REGION Network 114: NG_1
   RUNG wire#powerrail
      Contact( "AlwaysTRUE" )
      wire#w1
      Contact( "PalletNGData".LoadingNGPallet.NG_2_1 )
      Contact( "PalletNGData".LoadingNGPallet.NG_2_2 )
      Contact( "PalletNGData".LoadingNGPallet.NG_2_3 )
      Contact( "PalletNGData".LoadingNGPallet.NG_2_4 )
      Contact( "PalletNGData".LoadingNGPallet.NG_2_5 )
      { S7_Templates := "time_type := Time" } "TON".TON[50].TON(pt := t#4s, et =>)
      Coil( "ST10_DeviceError"."E".NG_1.ShaftScanNGFull )
   END_RUNG
   RUNG wire#w1
      Contact( "PalletNGData".LoadingNGPallet.NG_1_1 )
      Contact( "PalletNGData".LoadingNGPallet.NG_1_2 )
      Contact( "PalletNGData".LoadingNGPallet.NG_1_3 )
      Contact( "PalletNGData".LoadingNGPallet.NG_1_4 )
      Contact( "PalletNGData".LoadingNGPallet.NG_1_5 )
      { S7_Templates := "time_type := Time" } "TON".TON[51].TON(pt := t#4s, et =>)
      Coil( "ST10_DeviceError"."E".NG_1.PressNGFull )
   END_RUNG
   RUNG wire#w1
      Contact( "PalletNGData".LoadingNGPallet.NG_3_1 )
      Contact( "PalletNGData".LoadingNGPallet.NG_3_2 )
      Contact( "PalletNGData".LoadingNGPallet.NG_3_3 )
      Contact( "PalletNGData".LoadingNGPallet.NG_3_4 )
      Contact( "PalletNGData".LoadingNGPallet.NG_3_5 )
      { S7_Templates := "time_type := Time" } "TON".TON[52].TON(pt := t#4s, et =>)
      Coil( "ST10_DeviceError"."E".NG_1.RingScanNGFull )
   END_RUNG
   RUNG wire#w1
      I_Contact( "PalletNGData".LoadingNGPallet.Ready_1 )
      Contact( "Station_Sys".Auto.Mode )
      I_Contact( "KukaRobot1_CtrlDB".sROBtoPLC.User.Cycle.DO225_ScanPosInside )
      I_Contact( "KukaRobot1_CtrlDB".sROBtoPLC.User.Cycle.DO265_LoadNGInside )
      { S7_Templates := "time_type := Time" } "TON".TON[53].TON(pt := t#4s, et =>)
      I_Contact( true )
      Coil( "ST10_DeviceError"."E".NG_1.ShaftScanStatus )
   END_RUNG
   RUNG wire#w1
      I_Contact( "PalletNGData".LoadingNGPallet.Ready_2 )
      Contact( "Station_Sys".Auto.Mode )
      I_Contact( "KukaRobot1_CtrlDB".sROBtoPLC.User.Cycle.DO225_ScanPosInside )
      I_Contact( "KukaRobot1_CtrlDB".sROBtoPLC.User.Cycle.DO265_LoadNGInside )
      { S7_Templates := "time_type := Time" } "TON".TON[54].TON(pt := t#4s, et =>)
      I_Contact( true )
      Coil( "ST10_DeviceError"."E".NG_1.PressNGStatus )
   END_RUNG
   RUNG wire#w1
      I_Contact( "PalletNGData".LoadingNGPallet.Ready_3 )
      Contact( "Station_Sys".Auto.Mode )
      I_Contact( "KukaRobot1_CtrlDB".sROBtoPLC.User.Cycle.DO225_ScanPosInside )
      I_Contact( "KukaRobot1_CtrlDB".sROBtoPLC.User.Cycle.DO265_LoadNGInside )
      { S7_Templates := "time_type := Time" } "TON".TON[55].TON(pt := t#4s, et =>)
      I_Contact( true )
      Coil( "ST10_DeviceError"."E".NG_1.RingScanNGStatus )
   END_RUNG
   // the same network as SCL:
   "TON".TON[50].TON(IN := "AlwaysTRUE" AND "PalletNGData".LoadingNGPallet.NG_2_1 AND "PalletNGData".LoadingNGPallet.NG_2_2 AND "PalletNGData".LoadingNGPallet.NG_2_3 AND "PalletNGData".LoadingNGPallet.NG_2_4 AND "PalletNGData".LoadingNGPallet.NG_2_5,
                     PT := t#4s);
   "ST10_DeviceError"."E".NG_1.ShaftScanNGFull := "TON".TON[50].Q;
   "TON".TON[51].TON(IN := "AlwaysTRUE" AND "PalletNGData".LoadingNGPallet.NG_1_1 AND "PalletNGData".LoadingNGPallet.NG_1_2 AND "PalletNGData".LoadingNGPallet.NG_1_3 AND "PalletNGData".LoadingNGPallet.NG_1_4 AND "PalletNGData".LoadingNGPallet.NG_1_5,
                     PT := t#4s);
   "ST10_DeviceError"."E".NG_1.PressNGFull := "TON".TON[51].Q;
   "TON".TON[52].TON(IN := "AlwaysTRUE" AND "PalletNGData".LoadingNGPallet.NG_3_1 AND "PalletNGData".LoadingNGPallet.NG_3_2 AND "PalletNGData".LoadingNGPallet.NG_3_3 AND "PalletNGData".LoadingNGPallet.NG_3_4 AND "PalletNGData".LoadingNGPallet.NG_3_5,
                     PT := t#4s);
   "ST10_DeviceError"."E".NG_1.RingScanNGFull := "TON".TON[52].Q;
   "TON".TON[53].TON(IN := "AlwaysTRUE" AND NOT "PalletNGData".LoadingNGPallet.Ready_1 AND "Station_Sys".Auto.Mode AND NOT "KukaRobot1_CtrlDB".sROBtoPLC.User.Cycle.DO225_ScanPosInside AND NOT "KukaRobot1_CtrlDB".sROBtoPLC.User.Cycle.DO265_LoadNGInside,
                     PT := t#4s);
   "ST10_DeviceError"."E".NG_1.ShaftScanStatus := "TON".TON[53].Q AND NOT true;
   "TON".TON[54].TON(IN := "AlwaysTRUE" AND NOT "PalletNGData".LoadingNGPallet.Ready_2 AND "Station_Sys".Auto.Mode AND NOT "KukaRobot1_CtrlDB".sROBtoPLC.User.Cycle.DO225_ScanPosInside AND NOT "KukaRobot1_CtrlDB".sROBtoPLC.User.Cycle.DO265_LoadNGInside,
                     PT := t#4s);
   "ST10_DeviceError"."E".NG_1.PressNGStatus := "TON".TON[54].Q AND NOT true;
   "TON".TON[55].TON(IN := "AlwaysTRUE" AND NOT "PalletNGData".LoadingNGPallet.Ready_3 AND "Station_Sys".Auto.Mode AND NOT "KukaRobot1_CtrlDB".sROBtoPLC.User.Cycle.DO225_ScanPosInside AND NOT "KukaRobot1_CtrlDB".sROBtoPLC.User.Cycle.DO265_LoadNGInside,
                     PT := t#4s);
   "ST10_DeviceError"."E".NG_1.RingScanNGStatus := "TON".TON[55].Q AND NOT true;
END_REGION

REGION Network 115: NG 1 Door NOT Closed
   RUNG wire#powerrail
      Contact( "AlwaysTRUE" )
      Contact( "Station_Sys".Auto.Mode )
      I_Contact( "oE-NG-01SafetyGate" )
      Coil( "ST10_DeviceError"."E".NG_1."NG 1 DoorOpen" )
   END_RUNG
   // the same network as SCL:
   "ST10_DeviceError"."E".NG_1."NG 1 DoorOpen" := "AlwaysTRUE" AND "Station_Sys".Auto.Mode AND NOT "oE-NG-01SafetyGate";
END_REGION

REGION Network 116: E NG_2
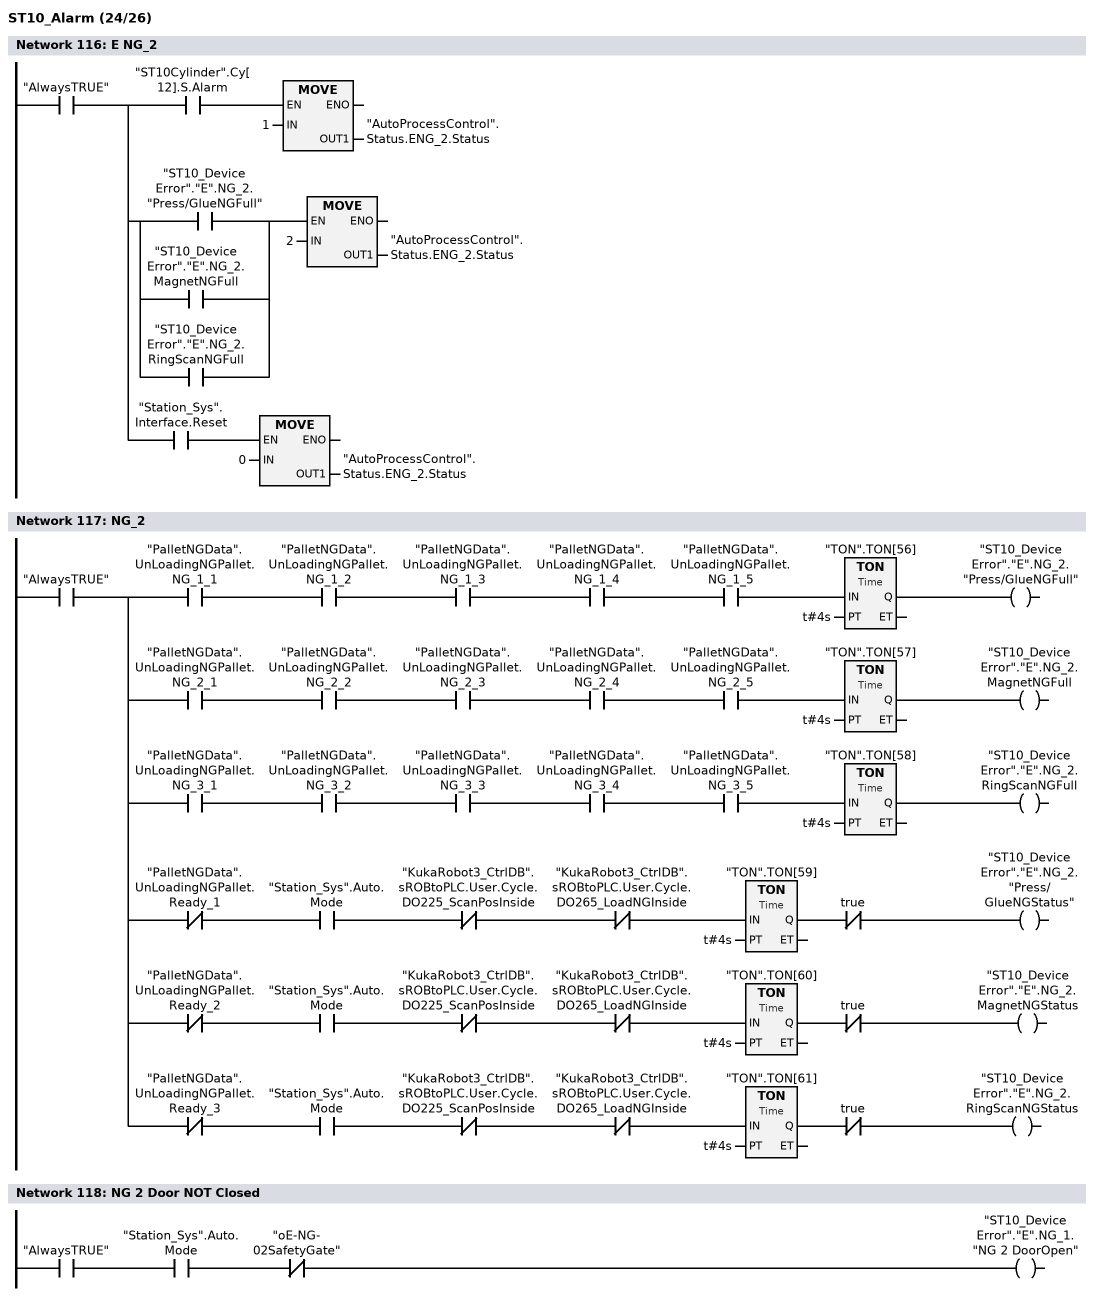
   RUNG wire#powerrail
      Contact( "AlwaysTRUE" )
      wire#w1
      Contact( "ST10Cylinder".Cy[12].S.Alarm )
      Move(in := 1, out1 => "AutoProcessControl".Status.ENG_2.Status)
   END_RUNG
   RUNG wire#w1
      Contact( "ST10_DeviceError"."E".NG_2."Press/GlueNGFull" )
      wire#w2
      Move(in := 2, out1 => "AutoProcessControl".Status.ENG_2.Status)
   END_RUNG
   RUNG wire#w1
      Contact( "ST10_DeviceError"."E".NG_2.MagnetNGFull )
   END_RUNG wire#w2
   RUNG wire#w1
      Contact( "ST10_DeviceError"."E".NG_2.RingScanNGFull )
   END_RUNG wire#w2
   RUNG wire#w1
      Contact( "Station_Sys".Interface.Reset )
      Move(in := 0, out1 => "AutoProcessControl".Status.ENG_2.Status)
   END_RUNG
   // the same network as SCL:
   IF "AlwaysTRUE" AND "ST10Cylinder".Cy[12].S.Alarm THEN
       "AutoProcessControl".Status.ENG_2.Status := 1;
   END_IF;
   IF "AlwaysTRUE" AND ("ST10_DeviceError"."E".NG_2."Press/GlueNGFull" OR "ST10_DeviceError"."E".NG_2.MagnetNGFull OR "ST10_DeviceError"."E".NG_2.RingScanNGFull) THEN
       "AutoProcessControl".Status.ENG_2.Status := 2;
   END_IF;
   IF "AlwaysTRUE" AND "Station_Sys".Interface.Reset THEN
       "AutoProcessControl".Status.ENG_2.Status := 0;
   END_IF;
END_REGION

REGION Network 117: NG_2
   RUNG wire#powerrail
      Contact( "AlwaysTRUE" )
      wire#w1
      Contact( "PalletNGData".UnLoadingNGPallet.NG_1_1 )
      Contact( "PalletNGData".UnLoadingNGPallet.NG_1_2 )
      Contact( "PalletNGData".UnLoadingNGPallet.NG_1_3 )
      Contact( "PalletNGData".UnLoadingNGPallet.NG_1_4 )
      Contact( "PalletNGData".UnLoadingNGPallet.NG_1_5 )
      { S7_Templates := "time_type := Time" } "TON".TON[56].TON(pt := t#4s, et =>)
      Coil( "ST10_DeviceError"."E".NG_2."Press/GlueNGFull" )
   END_RUNG
   RUNG wire#w1
      Contact( "PalletNGData".UnLoadingNGPallet.NG_2_1 )
      Contact( "PalletNGData".UnLoadingNGPallet.NG_2_2 )
      Contact( "PalletNGData".UnLoadingNGPallet.NG_2_3 )
      Contact( "PalletNGData".UnLoadingNGPallet.NG_2_4 )
      Contact( "PalletNGData".UnLoadingNGPallet.NG_2_5 )
      { S7_Templates := "time_type := Time" } "TON".TON[57].TON(pt := t#4s, et =>)
      Coil( "ST10_DeviceError"."E".NG_2.MagnetNGFull )
   END_RUNG
   RUNG wire#w1
      Contact( "PalletNGData".UnLoadingNGPallet.NG_3_1 )
      Contact( "PalletNGData".UnLoadingNGPallet.NG_3_2 )
      Contact( "PalletNGData".UnLoadingNGPallet.NG_3_3 )
      Contact( "PalletNGData".UnLoadingNGPallet.NG_3_4 )
      Contact( "PalletNGData".UnLoadingNGPallet.NG_3_5 )
      { S7_Templates := "time_type := Time" } "TON".TON[58].TON(pt := t#4s, et =>)
      Coil( "ST10_DeviceError"."E".NG_2.RingScanNGFull )
   END_RUNG
   RUNG wire#w1
      I_Contact( "PalletNGData".UnLoadingNGPallet.Ready_1 )
      Contact( "Station_Sys".Auto.Mode )
      I_Contact( "KukaRobot3_CtrlDB".sROBtoPLC.User.Cycle.DO225_ScanPosInside )
      I_Contact( "KukaRobot3_CtrlDB".sROBtoPLC.User.Cycle.DO265_LoadNGInside )
      { S7_Templates := "time_type := Time" } "TON".TON[59].TON(pt := t#4s, et =>)
      I_Contact( true )
      Coil( "ST10_DeviceError"."E".NG_2."Press/GlueNGStatus" )
   END_RUNG
   RUNG wire#w1
      I_Contact( "PalletNGData".UnLoadingNGPallet.Ready_2 )
      Contact( "Station_Sys".Auto.Mode )
      I_Contact( "KukaRobot3_CtrlDB".sROBtoPLC.User.Cycle.DO225_ScanPosInside )
      I_Contact( "KukaRobot3_CtrlDB".sROBtoPLC.User.Cycle.DO265_LoadNGInside )
      { S7_Templates := "time_type := Time" } "TON".TON[60].TON(pt := t#4s, et =>)
      I_Contact( true )
      Coil( "ST10_DeviceError"."E".NG_2.MagnetNGStatus )
   END_RUNG
   RUNG wire#w1
      I_Contact( "PalletNGData".UnLoadingNGPallet.Ready_3 )
      Contact( "Station_Sys".Auto.Mode )
      I_Contact( "KukaRobot3_CtrlDB".sROBtoPLC.User.Cycle.DO225_ScanPosInside )
      I_Contact( "KukaRobot3_CtrlDB".sROBtoPLC.User.Cycle.DO265_LoadNGInside )
      { S7_Templates := "time_type := Time" } "TON".TON[61].TON(pt := t#4s, et =>)
      I_Contact( true )
      Coil( "ST10_DeviceError"."E".NG_2.RingScanNGStatus )
   END_RUNG
   // the same network as SCL:
   "TON".TON[56].TON(IN := "AlwaysTRUE" AND "PalletNGData".UnLoadingNGPallet.NG_1_1 AND "PalletNGData".UnLoadingNGPallet.NG_1_2 AND "PalletNGData".UnLoadingNGPallet.NG_1_3 AND "PalletNGData".UnLoadingNGPallet.NG_1_4 AND "PalletNGData".UnLoadingNGPallet.NG_1_5,
                     PT := t#4s);
   "ST10_DeviceError"."E".NG_2."Press/GlueNGFull" := "TON".TON[56].Q;
   "TON".TON[57].TON(IN := "AlwaysTRUE" AND "PalletNGData".UnLoadingNGPallet.NG_2_1 AND "PalletNGData".UnLoadingNGPallet.NG_2_2 AND "PalletNGData".UnLoadingNGPallet.NG_2_3 AND "PalletNGData".UnLoadingNGPallet.NG_2_4 AND "PalletNGData".UnLoadingNGPallet.NG_2_5,
                     PT := t#4s);
   "ST10_DeviceError"."E".NG_2.MagnetNGFull := "TON".TON[57].Q;
   "TON".TON[58].TON(IN := "AlwaysTRUE" AND "PalletNGData".UnLoadingNGPallet.NG_3_1 AND "PalletNGData".UnLoadingNGPallet.NG_3_2 AND "PalletNGData".UnLoadingNGPallet.NG_3_3 AND "PalletNGData".UnLoadingNGPallet.NG_3_4 AND "PalletNGData".UnLoadingNGPallet.NG_3_5,
                     PT := t#4s);
   "ST10_DeviceError"."E".NG_2.RingScanNGFull := "TON".TON[58].Q;
   "TON".TON[59].TON(IN := "AlwaysTRUE" AND NOT "PalletNGData".UnLoadingNGPallet.Ready_1 AND "Station_Sys".Auto.Mode AND NOT "KukaRobot3_CtrlDB".sROBtoPLC.User.Cycle.DO225_ScanPosInside AND NOT "KukaRobot3_CtrlDB".sROBtoPLC.User.Cycle.DO265_LoadNGInside,
                     PT := t#4s);
   "ST10_DeviceError"."E".NG_2."Press/GlueNGStatus" := "TON".TON[59].Q AND NOT true;
   "TON".TON[60].TON(IN := "AlwaysTRUE" AND NOT "PalletNGData".UnLoadingNGPallet.Ready_2 AND "Station_Sys".Auto.Mode AND NOT "KukaRobot3_CtrlDB".sROBtoPLC.User.Cycle.DO225_ScanPosInside AND NOT "KukaRobot3_CtrlDB".sROBtoPLC.User.Cycle.DO265_LoadNGInside,
                     PT := t#4s);
   "ST10_DeviceError"."E".NG_2.MagnetNGStatus := "TON".TON[60].Q AND NOT true;
   "TON".TON[61].TON(IN := "AlwaysTRUE" AND NOT "PalletNGData".UnLoadingNGPallet.Ready_3 AND "Station_Sys".Auto.Mode AND NOT "KukaRobot3_CtrlDB".sROBtoPLC.User.Cycle.DO225_ScanPosInside AND NOT "KukaRobot3_CtrlDB".sROBtoPLC.User.Cycle.DO265_LoadNGInside,
                     PT := t#4s);
   "ST10_DeviceError"."E".NG_2.RingScanNGStatus := "TON".TON[61].Q AND NOT true;
END_REGION

REGION Network 118: NG 2 Door NOT Closed
   RUNG wire#powerrail
      Contact( "AlwaysTRUE" )
      Contact( "Station_Sys".Auto.Mode )
      I_Contact( "oE-NG-02SafetyGate" )
      Coil( "ST10_DeviceError"."E".NG_1."NG 2 DoorOpen" )
   END_RUNG
   // the same network as SCL:
   "ST10_DeviceError"."E".NG_1."NG 2 DoorOpen" := "AlwaysTRUE" AND "Station_Sys".Auto.Mode AND NOT "oE-NG-02SafetyGate";
END_REGION

REGION Network 119: Press1
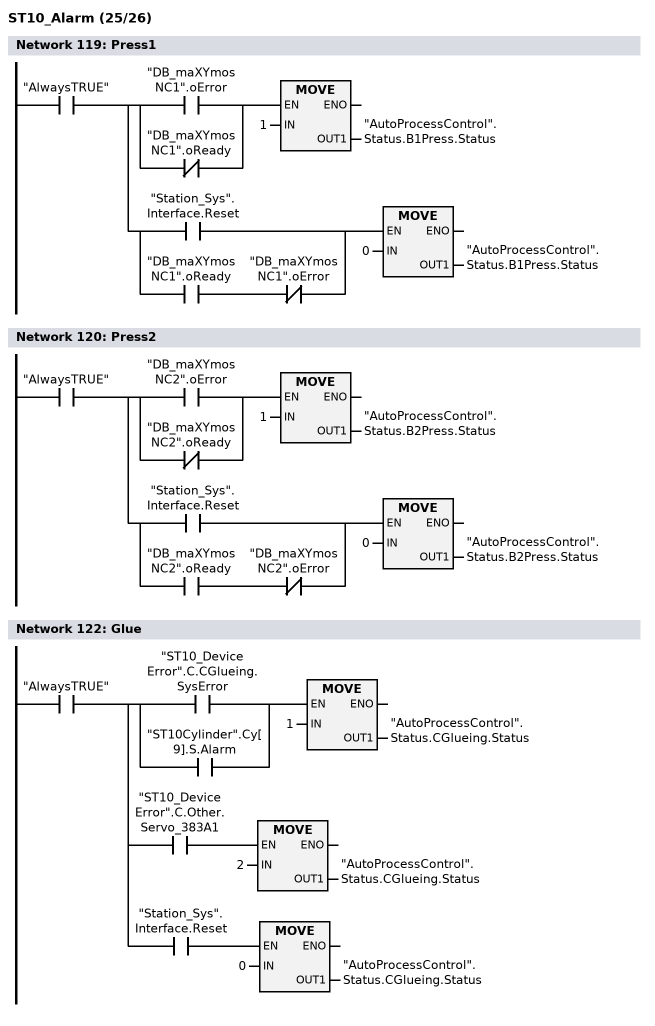
   RUNG wire#powerrail
      Contact( "AlwaysTRUE" )
      wire#w1
      Contact( "DB_maXYmosNC1".oError )
      wire#w2
      Move(in := 1, out1 => "AutoProcessControl".Status.B1Press.Status)
   END_RUNG
   RUNG wire#w1
      I_Contact( "DB_maXYmosNC1".oReady )
   END_RUNG wire#w2
   RUNG wire#w1
      Contact( "Station_Sys".Interface.Reset )
      wire#w3
      Move(in := 0, out1 => "AutoProcessControl".Status.B1Press.Status)
   END_RUNG
   RUNG wire#w1
      Contact( "DB_maXYmosNC1".oReady )
      I_Contact( "DB_maXYmosNC1".oError )
   END_RUNG wire#w3
   // the same network as SCL:
   IF "AlwaysTRUE" AND ("DB_maXYmosNC1".oError OR NOT "DB_maXYmosNC1".oReady) THEN
       "AutoProcessControl".Status.B1Press.Status := 1;
   END_IF;
   IF "AlwaysTRUE" AND ("Station_Sys".Interface.Reset OR ("DB_maXYmosNC1".oReady AND NOT "DB_maXYmosNC1".oError)) THEN
       "AutoProcessControl".Status.B1Press.Status := 0;
   END_IF;
END_REGION

REGION Network 120: Press2
   RUNG wire#powerrail
      Contact( "AlwaysTRUE" )
      wire#w1
      Contact( "DB_maXYmosNC2".oError )
      wire#w2
      Move(in := 1, out1 => "AutoProcessControl".Status.B2Press.Status)
   END_RUNG
   RUNG wire#w1
      I_Contact( "DB_maXYmosNC2".oReady )
   END_RUNG wire#w2
   RUNG wire#w1
      Contact( "Station_Sys".Interface.Reset )
      wire#w3
      Move(in := 0, out1 => "AutoProcessControl".Status.B2Press.Status)
   END_RUNG
   RUNG wire#w1
      Contact( "DB_maXYmosNC2".oReady )
      I_Contact( "DB_maXYmosNC2".oError )
   END_RUNG wire#w3
   // the same network as SCL:
   IF "AlwaysTRUE" AND ("DB_maXYmosNC2".oError OR NOT "DB_maXYmosNC2".oReady) THEN
       "AutoProcessControl".Status.B2Press.Status := 1;
   END_IF;
   IF "AlwaysTRUE" AND ("Station_Sys".Interface.Reset OR ("DB_maXYmosNC2".oReady AND NOT "DB_maXYmosNC2".oError)) THEN
       "AutoProcessControl".Status.B2Press.Status := 0;
   END_IF;
END_REGION

REGION Network 121: ******************** Glue ********************
END_REGION

REGION Network 122: Glue
   RUNG wire#powerrail
      Contact( "AlwaysTRUE" )
      wire#w1
      Contact( "ST10_DeviceError".C.CGlueing.SysError )
      wire#w2
      Move(in := 1, out1 => "AutoProcessControl".Status.CGlueing.Status)
   END_RUNG
   RUNG wire#w1
      Contact( "ST10Cylinder".Cy[9].S.Alarm )
   END_RUNG wire#w2
   RUNG wire#w1
      Contact( "ST10_DeviceError".C.Other.Servo_383A1 )
      Move(in := 2, out1 => "AutoProcessControl".Status.CGlueing.Status)
   END_RUNG
   RUNG wire#w1
      Contact( "Station_Sys".Interface.Reset )
      Move(in := 0, out1 => "AutoProcessControl".Status.CGlueing.Status)
   END_RUNG
   // the same network as SCL:
   IF "AlwaysTRUE" AND ("ST10_DeviceError".C.CGlueing.SysError OR "ST10Cylinder".Cy[9].S.Alarm) THEN
       "AutoProcessControl".Status.CGlueing.Status := 1;
   END_IF;
   IF "AlwaysTRUE" AND "ST10_DeviceError".C.Other.Servo_383A1 THEN
       "AutoProcessControl".Status.CGlueing.Status := 2;
   END_IF;
   IF "AlwaysTRUE" AND "Station_Sys".Interface.Reset THEN
       "AutoProcessControl".Status.CGlueing.Status := 0;
   END_IF;
END_REGION

REGION Network 123: A1 Table
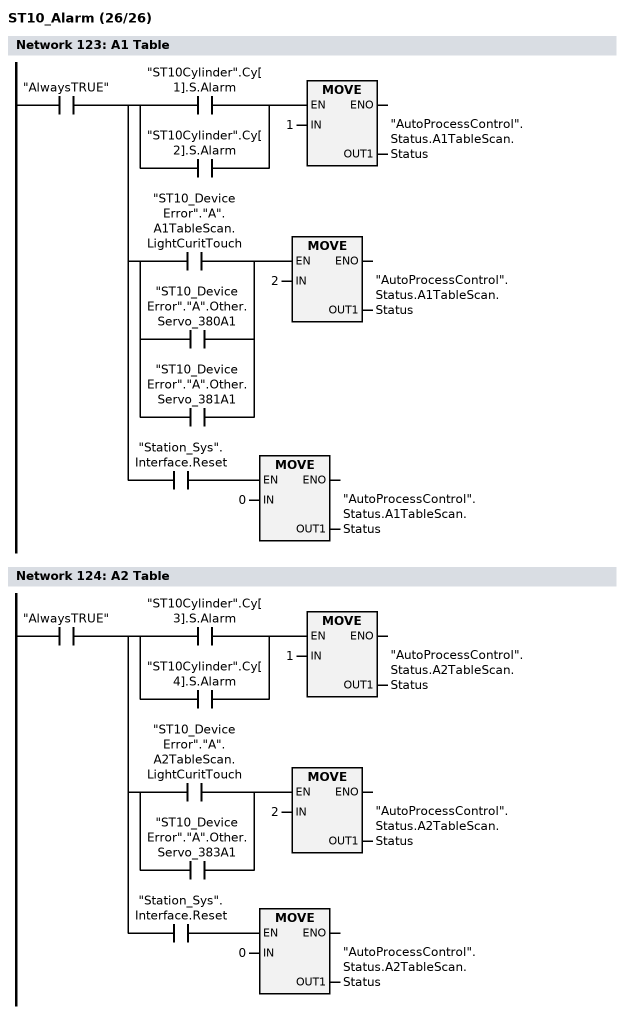
   RUNG wire#powerrail
      Contact( "AlwaysTRUE" )
      wire#w1
      Contact( "ST10Cylinder".Cy[1].S.Alarm )
      wire#w2
      Move(in := 1, out1 => "AutoProcessControl".Status.A1TableScan.Status)
   END_RUNG
   RUNG wire#w1
      Contact( "ST10Cylinder".Cy[2].S.Alarm )
   END_RUNG wire#w2
   RUNG wire#w1
      Contact( "ST10_DeviceError"."A".A1TableScan.LightCuritTouch )
      wire#w3
      Move(in := 2, out1 => "AutoProcessControl".Status.A1TableScan.Status)
   END_RUNG
   RUNG wire#w1
      Contact( "ST10_DeviceError"."A".Other.Servo_380A1 )
   END_RUNG wire#w3
   RUNG wire#w1
      Contact( "ST10_DeviceError"."A".Other.Servo_381A1 )
   END_RUNG wire#w3
   RUNG wire#w1
      Contact( "Station_Sys".Interface.Reset )
      Move(in := 0, out1 => "AutoProcessControl".Status.A1TableScan.Status)
   END_RUNG
   // the same network as SCL:
   IF "AlwaysTRUE" AND ("ST10Cylinder".Cy[1].S.Alarm OR "ST10Cylinder".Cy[2].S.Alarm) THEN
       "AutoProcessControl".Status.A1TableScan.Status := 1;
   END_IF;
   IF "AlwaysTRUE" AND ("ST10_DeviceError"."A".A1TableScan.LightCuritTouch OR "ST10_DeviceError"."A".Other.Servo_380A1 OR "ST10_DeviceError"."A".Other.Servo_381A1) THEN
       "AutoProcessControl".Status.A1TableScan.Status := 2;
   END_IF;
   IF "AlwaysTRUE" AND "Station_Sys".Interface.Reset THEN
       "AutoProcessControl".Status.A1TableScan.Status := 0;
   END_IF;
END_REGION

REGION Network 124: A2 Table
   RUNG wire#powerrail
      Contact( "AlwaysTRUE" )
      wire#w1
      Contact( "ST10Cylinder".Cy[3].S.Alarm )
      wire#w2
      Move(in := 1, out1 => "AutoProcessControl".Status.A2TableScan.Status)
   END_RUNG
   RUNG wire#w1
      Contact( "ST10Cylinder".Cy[4].S.Alarm )
   END_RUNG wire#w2
   RUNG wire#w1
      Contact( "ST10_DeviceError"."A".A2TableScan.LightCuritTouch )
      wire#w3
      Move(in := 2, out1 => "AutoProcessControl".Status.A2TableScan.Status)
   END_RUNG
   RUNG wire#w1
      Contact( "ST10_DeviceError"."A".Other.Servo_383A1 )
   END_RUNG wire#w3
   RUNG wire#w1
      Contact( "Station_Sys".Interface.Reset )
      Move(in := 0, out1 => "AutoProcessControl".Status.A2TableScan.Status)
   END_RUNG
   // the same network as SCL:
   IF "AlwaysTRUE" AND ("ST10Cylinder".Cy[3].S.Alarm OR "ST10Cylinder".Cy[4].S.Alarm) THEN
       "AutoProcessControl".Status.A2TableScan.Status := 1;
   END_IF;
   IF "AlwaysTRUE" AND ("ST10_DeviceError"."A".A2TableScan.LightCuritTouch OR "ST10_DeviceError"."A".Other.Servo_383A1) THEN
       "AutoProcessControl".Status.A2TableScan.Status := 2;
   END_IF;
   IF "AlwaysTRUE" AND "Station_Sys".Interface.Reset THEN
       "AutoProcessControl".Status.A2TableScan.Status := 0;
   END_IF;
END_REGION
END_FUNCTION
